// TIA Portal V20 export
// export: Created 2025-12-01T14:57:19.2912749Z, ExportSetting None, DisplayName Totally Integrated Automation Portal, DisplayVersion V20 Update 3, DisplayName TIA Portal Openness, DisplayVersion V20 Update 3, DisplayName TIA Portal Version Control Interface, DisplayVersion V20 Update 3, DisplayName STEP 7 Professional, DisplayVersion V20 Update 3, DisplayName STEP 7 Safety, DisplayVersion V20 Update 2, DisplayName WinCC Basic/Comfort/Advanced, DisplayVersion V20 Update 3, DisplayName WinCC Professional, DisplayVersion V20 Update 3, DisplayName WinCC Unified, DisplayVersion V20 Update 3
DATA_BLOCK "DB919_Temporizadores_Registro_flujos"   // DB919
{ S7_Optimized_Access := 'TRUE' }
// stored: AutoNumber false, MemoryReserve 0
   VAR
      Temporizadores_mesa { S7_SetPoint := 'True'} : Array[1.."CTE_MaxMesas"] of "Temporizadores_flujos_mesa";
   END_VAR
BEGIN
END_DATA_BLOCK
